FUNCTION_BLOCK MatrixInverse2x2 (* Basic FB with empty ECC *)
  (* Standard: 61499-2 *)
  (* Version 1.0, 2020-07-23, Candra Wardaya, UGM *)
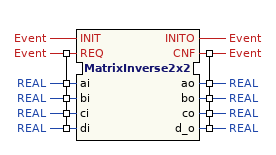
  EVENT_INPUT
    INIT; (* Initial Input *)
    REQ WITH ai, bi, ci, di; (* Execution Request *)
  END_EVENT
  EVENT_OUTPUT
    INITO; (* Initial Output *)
    CNF WITH ao, bo, co, d_o; (* Confirmation *)
  END_EVENT
  VAR_INPUT
    ai : REAL; (* Single real input *)
    bi : REAL; (* Single real input *)
    ci : REAL; (* Single real input *)
    di : REAL; (* Single real input *)
  END_VAR
  VAR_OUTPUT
    ao : REAL; (* Single real output *)
    bo : REAL; (* Single real output *)
    co : REAL; (* Single real output *)
    d_o : REAL; (* Single real output *)
  END_VAR
  VAR
    det : REAL; (* Determinant *)
  END_VAR
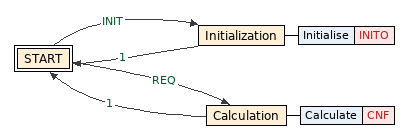
  EC_STATES
    START; (* Initial State *)
    Initialization : Initialise -> INITO;
    Calculation : Calculate -> CNF;
  END_STATES
  EC_TRANSITIONS
    START TO Initialization := INIT;
    Initialization TO START := 1;
    START TO Calculation := REQ;
    Calculation TO START := 1;
  END_TRANSITIONS
  ALGORITHM Calculate IN ST: (* New Algorithm *)
det := 1/(ai*di - ci*bi);  //determinant

ao := di*det;
bo := -bi*det;
co := -ci*det;
d_o := ai*det;
  END_ALGORITHM
  ALGORITHM Initialise IN ST: (* New Algorithm *)

  END_ALGORITHM
END_FUNCTION_BLOCK
